Omron Sysmac Studio project Pnomatik_Pick_Place_Uygulamasi (Sysmac Studio 1.65.0.64007, StandardProject)

# Controller new_Controller_0: NX1P2-1040DT1 version 1.69
Task PrimaryTask (priority 4, period or condition 2000): Program0

VAR_GLOBAL
    IN_Start_Button : BOOL;
    IN_Stop_Button : BOOL;
    IN_Urun_Alma_Sens : BOOL;
    IN_Urun_Tutucu_Sens : BOOL;
    IN_Urun_Yerlestirme_Sens : BOOL;
    IN_Reset_Button : BOOL;
    OUT_Konveyor1 : BOOL;
    OUT_Konveyor2 : BOOL;
    OUT_Tutucu_Valf : BOOL;
    OUT_Z_Valf : BOOL;
    OUT_X_Valf : BOOL;
END_VAR

PROGRAM Program0
VAR
    Start : BOOL;
    TON1 : TON;
    TON2 : TON;
    TON3 : TON;
    TON4 : TON;
    Kutu_Sayisi : INT;
    Adim : INT;
    TON5 : TON;
    TON6 : TON;
    TON7 : TON;
    TON8 : TON;
END_VAR
VAR_EXTERNAL
    IN_Start_Button : BOOL;
    IN_Stop_Button : BOOL;
    IN_Urun_Alma_Sens : BOOL;
    OUT_Konveyor1 : BOOL;
    OUT_Konveyor2 : BOOL;
    IN_Urun_Yerlestirme_Sens : BOOL;
    IN_Reset_Button : BOOL;
    OUT_Z_Valf : BOOL;
    IN_Urun_Tutucu_Sens : BOOL;
    OUT_Tutucu_Valf : BOOL;
    OUT_X_Valf : BOOL;
END_VAR
VAR
    _e1 : R_TRIG;
    _e2 : R_TRIG;
    _e3 : R_TRIG;
    _e4 : R_TRIG;
    _e5 : F_TRIG;
    _e6 : R_TRIG;
END_VAR

(* Section Section0: ladder, written here as Structured Text *)

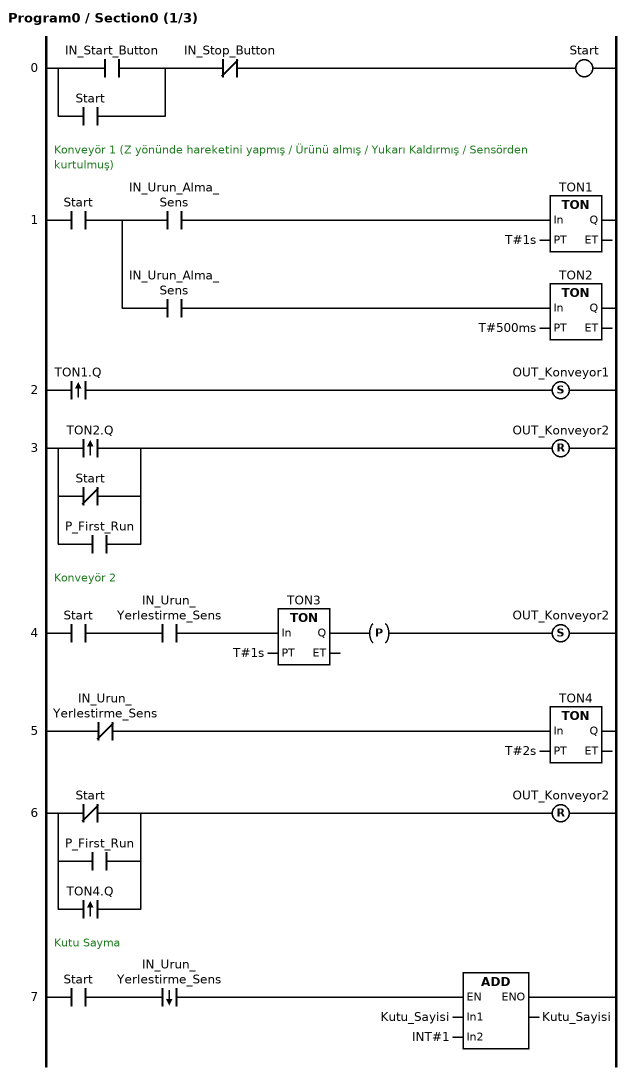
(* Rung 0 *)
Start := (IN_Start_Button OR Start) AND NOT IN_Stop_Button;
(* Rung 1: Konveyör 1 (Z yönünde hareketini yapmış / Ürünü almış / Yukarı Kaldırmış / Sensörden kurtulmuş) *)
TON1(In := Start AND IN_Urun_Alma_Sens, PT := T#1s);
TON2(In := Start AND IN_Urun_Alma_Sens, PT := T#500ms);
(* Rung 2 *)
_e1(CLK := TON1.Q);
IF _e1.Q THEN OUT_Konveyor1 := TRUE; END_IF;
(* Rung 3 *)
_e2(CLK := TON2.Q);
IF _e2.Q OR NOT Start OR P_First_Run THEN OUT_Konveyor2 := FALSE; END_IF;
(* Rung 4: Konveyör 2 *)
TON3(In := Start AND IN_Urun_Yerlestirme_Sens, PT := T#1s);
_e3(CLK := TON3.Q);
IF _e3.Q THEN OUT_Konveyor2 := TRUE; END_IF;
(* Rung 5 *)
TON4(In := NOT IN_Urun_Yerlestirme_Sens, PT := T#2s);
(* Rung 6 *)
_e4(CLK := TON4.Q);
IF NOT Start OR P_First_Run OR _e4.Q THEN OUT_Konveyor2 := FALSE; END_IF;
(* Rung 7: Kutu Sayma *)
_e5(CLK := IN_Urun_Yerlestirme_Sens);
IF Start AND _e5.Q THEN Kutu_Sayisi := Kutu_Sayisi + INT#1; END_IF;

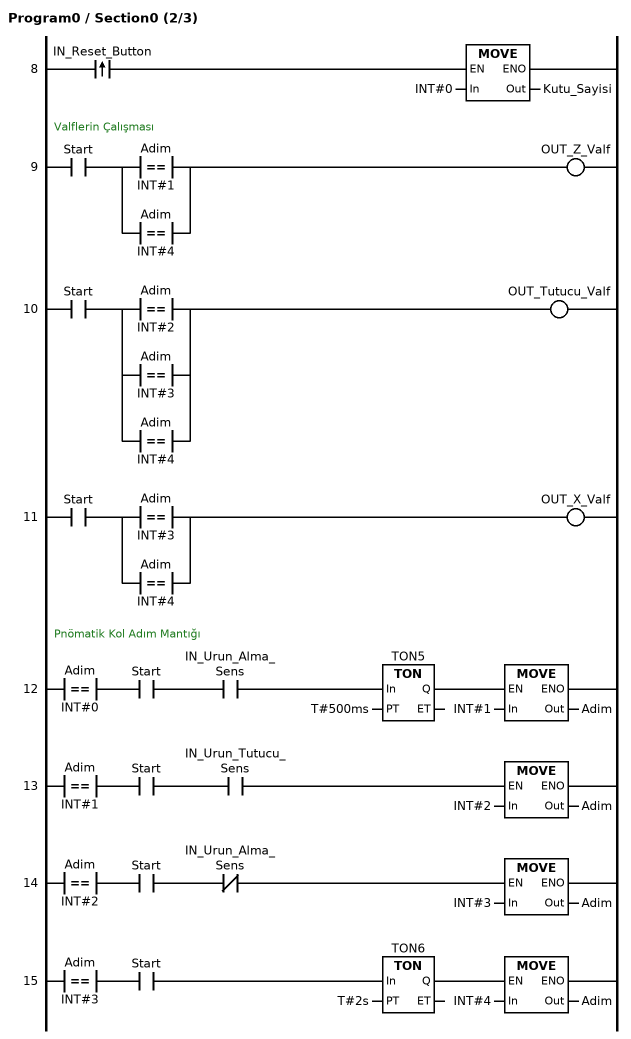
(* Rung 8 *)
_e6(CLK := IN_Reset_Button);
IF _e6.Q THEN Kutu_Sayisi := INT#0; END_IF;
(* Rung 9: Valflerin Çalışması *)
OUT_Z_Valf := Start AND ((Adim = INT#1) OR (Adim = INT#4));
(* Rung 10 *)
OUT_Tutucu_Valf := Start AND ((Adim = INT#2) OR (Adim = INT#3) OR (Adim = INT#4));
(* Rung 11 *)
OUT_X_Valf := Start AND ((Adim = INT#3) OR (Adim = INT#4));
(* Rung 12: Pnömatik Kol Adım Mantığı *)
TON5(In := (Adim = INT#0) AND Start AND IN_Urun_Alma_Sens, PT := T#500ms);
IF TON5.Q THEN Adim := INT#1; END_IF;
(* Rung 13 *)
IF (Adim = INT#1) AND Start AND IN_Urun_Tutucu_Sens THEN Adim := INT#2; END_IF;
(* Rung 14 *)
IF (Adim = INT#2) AND Start AND NOT IN_Urun_Alma_Sens THEN Adim := INT#3; END_IF;
(* Rung 15 *)
TON6(In := (Adim = INT#3) AND Start, PT := T#2s);
IF TON6.Q THEN Adim := INT#4; END_IF;

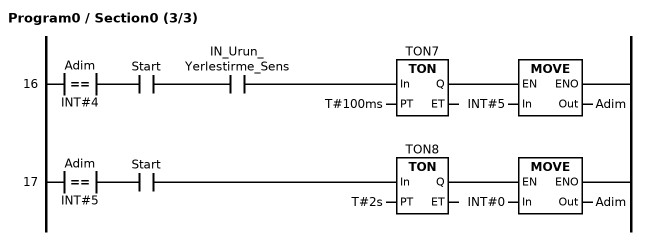
(* Rung 16 *)
TON7(In := (Adim = INT#4) AND Start AND IN_Urun_Yerlestirme_Sens, PT := T#100ms);
IF TON7.Q THEN Adim := INT#5; END_IF;
(* Rung 17 *)
TON8(In := (Adim = INT#5) AND Start, PT := T#2s);
IF TON8.Q THEN Adim := INT#0; END_IF;
END_PROGRAM